// TIA Portal V18 export
DATA_BLOCK "WN_0_root"   // DB7
VERSION : 0.1
// stored: AutoNumber true, DBAccessibleFromOPCUA true, InstanceOfName ER_WN__root_FB, InstanceOfType FB
"ER_WN__root_FB"
   // VAR_INPUT
   //    ER_count : Int;
   //    ACK : Bool;
   // END_VAR
   // VAR_OUTPUT
   //    ER_exists : Bool;
   // END_VAR
BEGIN
END_DATA_BLOCK
